{attribute 'linkalways'} 
{attribute 'no_explicit_call' := 'This FB is a CLASS and must be accessed using methods or properties'}
{attribute 'enable_dynamic_creation'}
{attribute 'TcRpcEnable'}
FUNCTION_BLOCK RpcServer IMPLEMENTS I_RpcServer
VAR
	// default header accessor.
	headerAccessor : HeaderAccessor;
	
	// Payload size may be changed using the constants
	payloadStringSizeIncludingNull : UDINT := ServerConfiguration.PAYLOAD_STRING_SIZE + 1;
	
	// the middleware stack allows us to construct our server in any way needed.
	// by default we will support sessions, async polling and chunked requests/
	middlewareStack : MiddlewareStack;
	
	// responseId generation required for pending or chunked data
	sequentialResponseIdGenerator : SequentialResponseIdGenerator;
	
	// ability to support sessions...
	sessionIdGenerator : SequentialSessionIdGenerator;
	sessionManager : SessionManager(sessionIdGenerator, INACTIVE_SESSION_MAX_AGE);
	sessionsMiddleware : SessionsMiddleware(sessionManager, headerAccessor);
	
	// ability to suppoort chunked requests
	chunkedRequestsManager : ChunkedRequestsManager(payloadStringSizeIncludingNull, sessionManager, headerAccessor);
	chunkedRequestsMiddleware : ChunkedRequestsMiddleware(chunkedRequestsManager);
	
	// ability to support chunked responses
	chunkedResponseManager : ChunkedResponseManager(payloadStringSizeIncludingNull, sessionManager, sequentialResponseIdGenerator, headerAccessor);
	chunkedResponsesMiddleware : ChunkedResponsesMiddleware(chunkedResponseManager);
	
	// ability to support pending responses
	asyncResponseManager : AsyncResponseManager(sessionManager, sequentialResponseIdGenerator, headerAccessor);
	asyncResponseMiddleware : AsyncResponseMiddleware(asyncResponseManager);
	
	// ability to support rpc
	synchronousRpcHandlers : SynchronousRpcHandlers;
	asynchronousRpcHandlers : AsynchronousRpcHandlers;
	asyncRpcCallQueue : AsyncRpcCallQueue;
	rpcManager : RpcManager(synchronousRpcHandlers, asynchronousRpcHandlers, asyncResponseManager, headerAccessor, asyncRpcCallQueue);
	rpcMiddleware : RpcMiddleware(rpcManager);
	
	// registered apis (used for cyclic calling)
	registeredRpcApis : RegisteredRpcApis;
	
END_VAR
VAR CONSTANT
	INACTIVE_SESSION_MAX_AGE : TIME := T#10S;
END_VAR

METHOD PUBLIC CyclicCall
VAR_INPUT
END_VAR
sessionManager.CyclicCall();
asyncRpcCallQueue.CyclicCall();
registeredRpcApis.CyclicCall();
END_METHOD

METHOD FB_init : BOOL
VAR_INPUT
	bInitRetains : BOOL; // if TRUE, the retain variables are initialized (warm start / cold start)
	bInCopyCode : BOOL;  // if TRUE, the instance afterwards gets moved into the copy code (online change)
END_VAR
// must be above any middleware which requires storing of session data. 
// best practice is to put at the top
MiddlewareStack.Use(sessionsMiddleware);

// must be above any middleware which could send a response larger than the max payload.
// once this is in place then middleware can send as large as they like (up to router memory max)
MiddlewareStack.Use(chunkedResponsesMiddleware);

// must be above any middleware which needs to support async responses
MiddlewareStack.Use(AsyncResponseMiddleware);

// chunked request must be after chunked response to prevent incorrectly starting a new request
// if the client askes for a response without removing the last request header.
MiddlewareStack.Use(chunkedRequestsMiddleware); 

// rpc middlware.  All other middleware can go under here.
MiddlewareStack.Use(rpcMiddleware);
END_METHOD

{attribute 'TcRpcEnable'}
METHOD PUBLIC HandleRequest : ResponseData;
VAR_INPUT
	SerializedHeader : STRING(ServerConfiguration.HEADER_STRING_SIZE);
	SerializedPayload : STRING(ServerConfiguration.PAYLOAD_STRING_SIZE);
END_VAR
VAR
	header : Header(SerializedHeader);
	request : Request(header, SerializedPayload);
	serverResponse : ServerResponse(headerAccessor);
END_VAR
middlewareStack.Handle(request, serverResponse);

IF NOT serverResponse.HeadersSent THEN
	serverResponse.Error('Unhandled Request');
END_IF

serverResponse.TryGetData(HandleRequest);
END_METHOD

METHOD PUBLIC RegisterApi
VAR_INPUT
	RpcApi : I_RpcApi;
END_VAR
RpcApi.RegisterSynchronousRpcHandlersWith(synchronousRpcHandlers);
RpcApi.RegisterAsynchronousRpcHandlersWith(asynchronousRpcHandlers);
registeredRpcApis.RegisterRpcApi(RpcApi);
END_METHOD

METHOD PUBLIC RegisterAsynchronousRpcHandler
VAR_INPUT
	MethodName : T_MAXSTRING;
	Handler : I_AsynchronousRpcHandler;
END_VAR
asynchronousRpcHandlers.RegisterHandler(MethodName, Handler);
END_METHOD

METHOD PUBLIC RegisterSynchronousRpcHandler
VAR_INPUT
	MethodName : T_MAXSTRING;
	Handler : I_SynchronousRpcHandler;
END_VAR
synchronousRpcHandlers.RegisterHandler(MethodName, Handler);
END_METHOD

PROPERTY PUBLIC SessionCount : DINT
GET
SessionCount := sessionManager.SessionCount;
END_GET
END_PROPERTY

METHOD PUBLIC Use
VAR_INPUT
	Middleware : I_Middleware;
END_VAR
middlewareStack.Use(Middleware);
END_METHOD

END_FUNCTION_BLOCK

(* stored: Version 1.1.0.1, ProductVersion 3.1.4024.12
   POU RpcServer: Id {d0c543ee-285c-0d92-3327-6786bf152970}, SpecialFunc None
   Folder Constructor: Id {cd2fe0ed-3f15-0d44-2e60-cbb6443221c1}
   Method CyclicCall: Id {539be5bf-e9a8-0ab6-0cd5-7dcc722256e0}
   Method FB_init: Id {76a0002b-f61d-0a35-104c-169abb3c3728}
   Method HandleRequest: Id {be6d2e0b-d137-0db3-37e1-f18d6e642bd1}
   Method RegisterApi: Id {562149a8-e0a7-4c1c-80dd-b24f63a0d991}
   Method RegisterAsynchronousRpcHandler: Id {f2c983c5-0460-0ac4-0ab1-c7c405c22fdf}
   Method RegisterSynchronousRpcHandler: Id {3f3f4dec-9dbc-41f8-98fa-f641cf39c9c1}
   Property SessionCount: Id {012b8c48-2d55-070c-2dc8-5f5a01686af8}
   Get Get: Id {ba5c5b9c-dd7d-09eb-32f7-db461311522c}
   Method Use: Id {5e295ea9-33ae-0561-0e53-6a8e1bcf642c} *)
